% RSLogix 500 project Project4-FINAL.RSS, saved by version 8.30.00.16 %
PROJECT "UNTITLED"    % processor: Bul.1763 MicroLogix 1100 Series B %

PROGRAM FILES
  LAD 2 "MAIN"  4 rungs
  LAD 3 "IO"  7 rungs
  LAD 4 "LOGIC"  11 rungs
  LAD 5 "POSITION"  10 rungs

DATA FILES
  O0 OUTPUT  5 elements
  I1 INPUT  7 elements
  S2 STATUS  66 elements
  B3 BINARY  3 elements
  T4 TIMER  3 elements
  C5 COUNTER  1 elements
  R6 CONTROL  1 elements
  N7 INTEGER  2 elements
  F8 FLOAT  1 elements

LADDER 2 "MAIN"
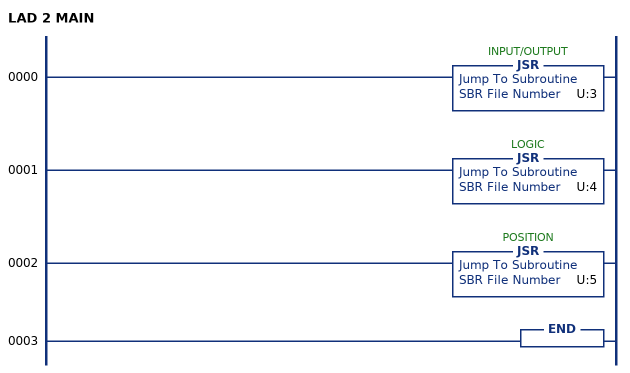
% Rung: 0 %
SOR JSR U:3 EOR
%   U:3  "INPUT/OUTPUT" %
% Rung: 1 %
SOR JSR U:4 EOR
%   U:4  "LOGIC" %
% Rung: 2 %
SOR JSR U:5 EOR
%   U:5  "POSITION" %
% Rung: 3 %
SOR END EOR

LADDER 3 "IO"
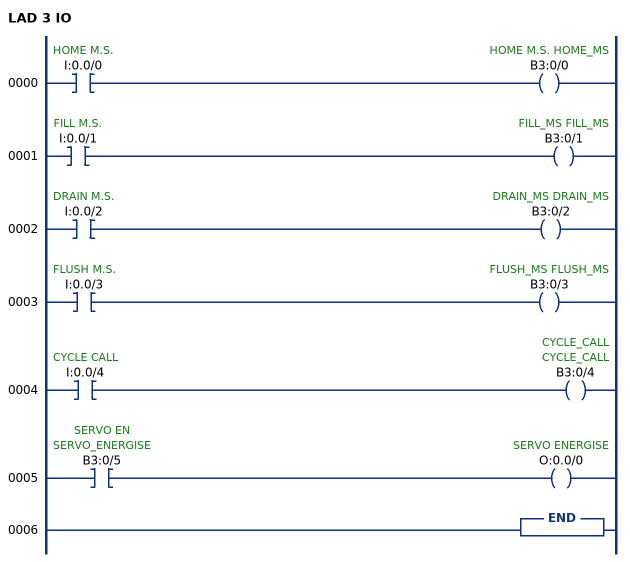
% Rung: 0 %
SOR XIC I:0.0/0 OTE B3:0/0 EOR
%   I:0.0/0  "HOME M.S." %
%   B3:0/0  HOME_MS  "HOME M.S." %
% Rung: 1 %
SOR XIC I:0.0/1 OTE B3:0/1 EOR
%   I:0.0/1  "FILL M.S." %
%   B3:0/1  FILL_MS  "FILL_MS" %
% Rung: 2 %
SOR XIC I:0.0/2 OTE B3:0/2 EOR
%   I:0.0/2  "DRAIN M.S." %
%   B3:0/2  DRAIN_MS  "DRAIN_MS" %
% Rung: 3 %
SOR XIC I:0.0/3 OTE B3:0/3 EOR
%   I:0.0/3  "FLUSH M.S." %
%   B3:0/3  FLUSH_MS  "FLUSH_MS" %
% Rung: 4 %
SOR XIC I:0.0/4 OTE B3:0/4 EOR
%   I:0.0/4  "CYCLE CALL" %
%   B3:0/4  CYCLE_CALL  "CYCLE_CALL" %
% Rung: 5 %
SOR XIC B3:0/5 OTE O:0.0/0 EOR
%   B3:0/5  SERVO_ENERGISE  "SERVO EN" %
%   O:0.0/0  "SERVO ENERGISE" %
% Rung: 6 %
SOR END EOR

LADDER 4 "LOGIC"
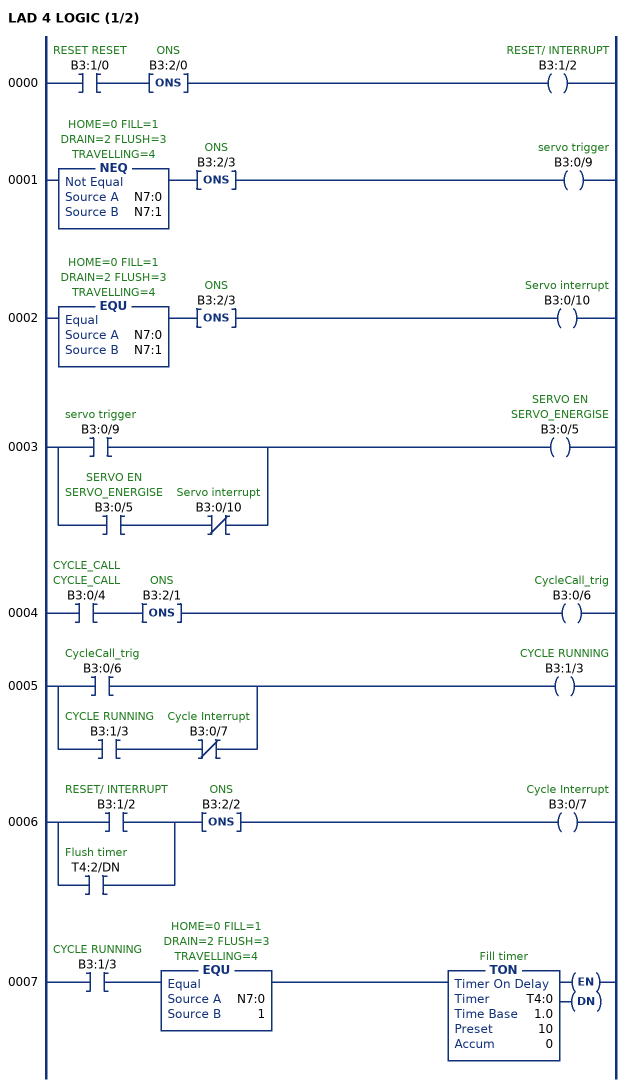
% Rung: 0 %
SOR XIC B3:1/0 ONS B3:2/0 OTE B3:1/2 EOR
%   B3:1/0  RESET  "RESET" %
%   B3:2/0  "ONS" %
%   B3:1/2  "RESET/ INTERRUPT" %
% Rung: 1 %
SOR NEQ N7:0 N7:1 ONS B3:2/3 OTE B3:0/9 EOR
%   N7:0  "HOME=0 FILL=1 DRAIN=2 FLUSH=3 TRAVELLING=4" %
%   N7:1  "DESIRED: HOME=0 FILL=1 DRAIN=2 FLUSH=3" %
%   B3:2/3  "ONS" %
%   B3:0/9  "servo trigger" %
% Rung: 2 %
SOR EQU N7:0 N7:1 ONS B3:2/3 OTE B3:0/10 EOR
%   N7:0  "HOME=0 FILL=1 DRAIN=2 FLUSH=3 TRAVELLING=4" %
%   N7:1  "DESIRED: HOME=0 FILL=1 DRAIN=2 FLUSH=3" %
%   B3:2/3  "ONS" %
%   B3:0/10  "Servo interrupt" %
% Rung: 3 %
SOR BST XIC B3:0/9 NXB XIC B3:0/5 XIO B3:0/10 BND OTE B3:0/5 EOR
%   B3:0/9  "servo trigger" %
%   B3:0/5  SERVO_ENERGISE  "SERVO EN" %
%   B3:0/10  "Servo interrupt" %
% Rung: 4 %
SOR XIC B3:0/4 ONS B3:2/1 OTE B3:0/6 EOR
%   B3:0/4  CYCLE_CALL  "CYCLE_CALL" %
%   B3:2/1  "ONS" %
%   B3:0/6  "CycleCall_trig" %
% Rung: 5 %
SOR BST XIC B3:0/6 NXB XIC B3:1/3 XIO B3:0/7 BND OTE B3:1/3 EOR
%   B3:0/6  "CycleCall_trig" %
%   B3:1/3  "CYCLE RUNNING" %
%   B3:0/7  "Cycle Interrupt" %
% Rung: 6 %
SOR BST XIC B3:1/2 NXB XIC T4:2/DN BND ONS B3:2/2 OTE B3:0/7 EOR
%   B3:1/2  "RESET/ INTERRUPT" %
%   T4:2  "Flush timer" %
%   B3:2/2  "ONS" %
%   B3:0/7  "Cycle Interrupt" %
% Rung: 7 %
SOR XIC B3:1/3 EQU N7:0 1 TON T4:0 1.0 10 0 EOR
%   B3:1/3  "CYCLE RUNNING" %
%   N7:0  "HOME=0 FILL=1 DRAIN=2 FLUSH=3 TRAVELLING=4" %
%   T4:0  "Fill timer" %

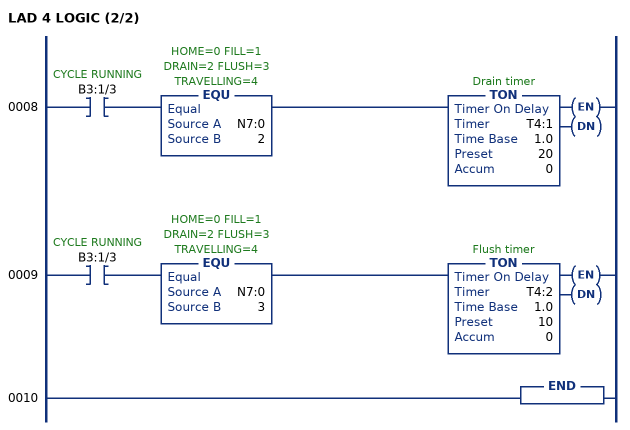
% Rung: 8 %
SOR XIC B3:1/3 EQU N7:0 2 TON T4:1 1.0 20 0 EOR
%   B3:1/3  "CYCLE RUNNING" %
%   N7:0  "HOME=0 FILL=1 DRAIN=2 FLUSH=3 TRAVELLING=4" %
%   T4:1  "Drain timer" %
% Rung: 9 %
SOR XIC B3:1/3 EQU N7:0 3 TON T4:2 1.0 10 0 EOR
%   B3:1/3  "CYCLE RUNNING" %
%   N7:0  "HOME=0 FILL=1 DRAIN=2 FLUSH=3 TRAVELLING=4" %
%   T4:2  "Flush timer" %
% Rung: 10 %
SOR END EOR

LADDER 5 "POSITION"
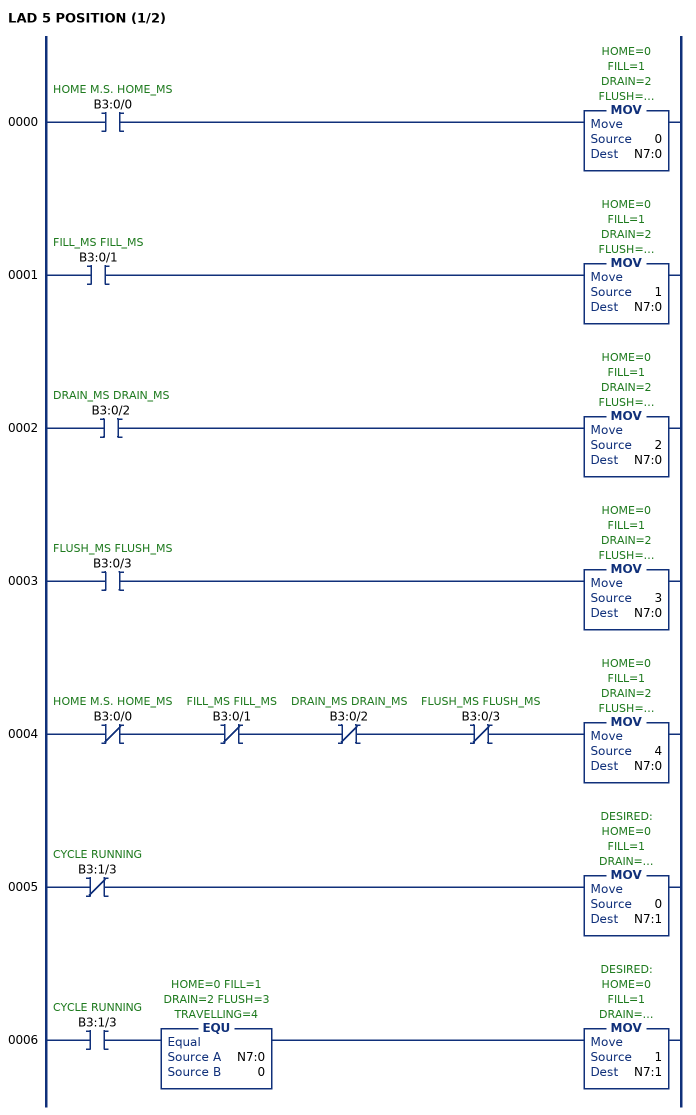
% Rung: 0 %
SOR XIC B3:0/0 MOV 0 N7:0 EOR
%   B3:0/0  HOME_MS  "HOME M.S." %
%   N7:0  "HOME=0 FILL=1 DRAIN=2 FLUSH=3 TRAVELLING=4" %
% Rung: 1 %
SOR XIC B3:0/1 MOV 1 N7:0 EOR
%   B3:0/1  FILL_MS  "FILL_MS" %
%   N7:0  "HOME=0 FILL=1 DRAIN=2 FLUSH=3 TRAVELLING=4" %
% Rung: 2 %
SOR XIC B3:0/2 MOV 2 N7:0 EOR
%   B3:0/2  DRAIN_MS  "DRAIN_MS" %
%   N7:0  "HOME=0 FILL=1 DRAIN=2 FLUSH=3 TRAVELLING=4" %
% Rung: 3 %
SOR XIC B3:0/3 MOV 3 N7:0 EOR
%   B3:0/3  FLUSH_MS  "FLUSH_MS" %
%   N7:0  "HOME=0 FILL=1 DRAIN=2 FLUSH=3 TRAVELLING=4" %
% Rung: 4 %
SOR XIO B3:0/0 XIO B3:0/1 XIO B3:0/2 XIO B3:0/3 MOV 4 N7:0 EOR
%   B3:0/0  HOME_MS  "HOME M.S." %
%   B3:0/1  FILL_MS  "FILL_MS" %
%   B3:0/2  DRAIN_MS  "DRAIN_MS" %
%   B3:0/3  FLUSH_MS  "FLUSH_MS" %
%   N7:0  "HOME=0 FILL=1 DRAIN=2 FLUSH=3 TRAVELLING=4" %
% Rung: 5 %
SOR XIO B3:1/3 MOV 0 N7:1 EOR
%   B3:1/3  "CYCLE RUNNING" %
%   N7:1  "DESIRED: HOME=0 FILL=1 DRAIN=2 FLUSH=3" %
% Rung: 6 %
SOR XIC B3:1/3 EQU N7:0 0 MOV 1 N7:1 EOR
%   B3:1/3  "CYCLE RUNNING" %
%   N7:0  "HOME=0 FILL=1 DRAIN=2 FLUSH=3 TRAVELLING=4" %
%   N7:1  "DESIRED: HOME=0 FILL=1 DRAIN=2 FLUSH=3" %

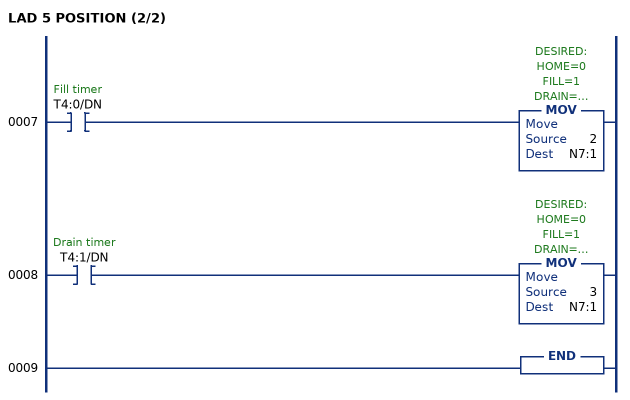
% Rung: 7 %
SOR XIC T4:0/DN MOV 2 N7:1 EOR
%   T4:0  "Fill timer" %
%   N7:1  "DESIRED: HOME=0 FILL=1 DRAIN=2 FLUSH=3" %
% Rung: 8 %
SOR XIC T4:1/DN MOV 3 N7:1 EOR
%   T4:1  "Drain timer" %
%   N7:1  "DESIRED: HOME=0 FILL=1 DRAIN=2 FLUSH=3" %
% Rung: 9 %
SOR END EOR

OTHER DOCUMENTED ADDRESSES
  B3:0/8  "Cycle Complete"
  B3:1/1  "RESET TRIG"

DATA TABLE (non-zero values as saved)
DATA T4
% .PRE .ACC %
% T4:0 % 10 0
% T4:1 % 20 0
% T4:2 % 10 0
